TYPE dutPul :
STRUCT
	xPul:BOOL;		// IN Pulsador
	xPil:BOOL;		// OUT Piloto

END_STRUCT
END_TYPE

(* stored: Version 1.1.0.1, ProductVersion 3.1.4024.10
   DUT dutPul: Id {b51280c3-2042-413a-a298-d7cbcc88d01e} *)
